PROGRAM PRG_ADS_Gauges
VAR
    {attribute 'pytmc' :=' pv: CRIXS:TM2K2:GCC:01 '}
    TM2K2_GCC_Reader : FB_TGCC_ADS;

    //{attribute 'pytmc' :=' pv: CRIXS:AT3K2:GCC:01 '}
    //AT3K2_GCC_Reader : FB_TGCC_ADS;

    // This variable needs to be instantiated for the Watchdog to work
    ADS_connection_counter : UDINT;
END_VAR

TM2K2_GCC_Reader(
    sNetId := '172.21.140.69.1.1', // plc-kfe-rix-vac
    nPort := 851, // ADS port of the PLC reading from this PLC
    sVarName := 'PRG_KFE_RIX_VAC.fb_TM2K2_K2B_GCC_1', // Full name of the FB containing the gauge to be read
    iWatchdog := ADS_connection_counter // UDINT required for watchdog functionality
);

//AT3K2_GCC_Reader(
//    sNetId := '172.21.140.69.1.1', // plc-kfe-rix-vac
//    nPort := 851, // ADS port of the PLC reading from this PLC
//    sVarName := 'PRG_KFE_RIX_VAC.fb_AT3K2_SOLID_GCC_1', // Full name of the FB containing the gauge to be read
//    iWatchdog := ADS_connection_counter // UDINT required for watchdog functionality
//);

END_PROGRAM

(* stored: Version 1.1.0.1, ProductVersion 3.1.4022.18
   POU PRG_ADS_Gauges: Id {987f64de-7f79-4420-9e0c-b19649a7caa1}, SpecialFunc None *)
